PROGRAM SerialCommunicationController
VAR
	// Handlers to call
	HandleSerialCommunication : SerialDataHandler;
	
	// Local variables
	_serialCommSetpoints : ST_SerialCommSetpoints;
	_serialCommReadData : ST_SerialCommReadData;
END_VAR


HandleSerialCommunication(
						serialCommSetpoints => _serialCommSetpoints,
						serialCommReadData => _serialCommReadData);

PROPERTY SerialCommReadData : ST_SerialCommReadData
GET

SerialCommReadData := _serialCommReadData;
END_GET
END_PROPERTY

PROPERTY SerialCommSetpoints : ST_SerialCommSetpoints
SET

_serialCommSetpoints := SerialCommSetpoints;
END_SET
END_PROPERTY

END_PROGRAM

(* stored: Version 1.1.0.1, ProductVersion 3.1.4024.9
   POU SerialCommunicationController: Id {a12e14a2-3147-4be8-a768-485775d9f2f3}, SpecialFunc None
   Property SerialCommReadData: Id {d42acb96-3051-4cc7-8cb4-b52d07a7c56e}
   Get Get: Id {105c5e16-d13b-4fb0-aa53-f0fcec0675c4}
   Property SerialCommSetpoints: Id {4e41ad63-edad-44ba-93f9-12f80b085bc1}
   Set Set: Id {5976fbf0-0c84-4fcb-9fc5-5b4c8068c325} *)
